FUNCTION_BLOCK SKILL_Chain (* Status chain link: aggregates Busy/Held/Running along the skills of an equipment module *)
  (* Standard: 61499-2 *)
  (* Version 2.0, 2026-09-27, Project contributors, Filling cell reference model *)
  PACKAGE fillingcell;
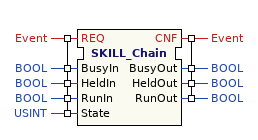
  EVENT_INPUT
    REQ WITH BusyIn, HeldIn, RunIn, State;
  END_EVENT
  EVENT_OUTPUT
    CNF WITH BusyOut, HeldOut, RunOut;
  END_EVENT
  VAR_INPUT
    BusyIn : BOOL;
    HeldIn : BOOL := TRUE;
    RunIn : BOOL := TRUE;
    State : USINT := 4;
  END_VAR
  VAR_OUTPUT
    BusyOut : BOOL;
    HeldOut : BOOL;
    RunOut : BOOL;
  END_VAR
  VAR
    MyBusy : BOOL;
  END_VAR
  EC_STATES
    REQ : REQ -> CNF;
  END_STATES
  ALGORITHM REQ IN ST:
MyBusy := NOT ((State = 4) OR (State = 17) OR (State = 2) OR (State = 9));
BusyOut := BusyIn OR MyBusy;
HeldOut := HeldIn AND ((NOT MyBusy) OR (State = 11));
RunOut := RunIn AND ((NOT MyBusy) OR (State = 6));
  END_ALGORITHM
END_FUNCTION_BLOCK
